INTERFACE I_Command EXTENDS I_Base

METHOD Execute : BOOL
VAR_INPUT
END_VAR
END_METHOD

END_INTERFACE

(* stored: Version 1.1.0.1, ProductVersion 3.1.4026.18
   Itf I_Command: Id {3e01d927-b142-422c-9639-5ff2d5ef7a2f}
   Method Execute: Id {731b3a30-6f02-445c-bb12-ffbfd0edf610} *)
